{attribute 'GeneratedUsingTerminal: EL6002-0000-0016'}
{attribute addProperty BoxType "EL6002-0000-0016"}
{attribute addProperty Id "EtcSlaveTerminalBaseCOM_Inputs_Channel_1AT %I*COM_Inputs_Channel_3801C95E30COM_Inputs_Channel_2AT %I*COM_Inputs_Channel_3801C95E30COM_Outputs_Channel_1AT %Q*COM_Outputs_Channel_EADA2E0D27COM_Outputs_Channel_2AT %Q*COM_Outputs_Channel_EADA2E0D27WcStateAT %I*WcState_9091E0EB2InfoDataAT %I*InfoData_32EB74EA10"}
{attribute addProperty CRC "2353564961"}
{attribute addProperty Size "126"}
TYPE EL6002_8C488D21 EXTENDS EtcSlaveTerminalBase :
STRUCT
	{attribute addProperty Name "COM_Inputs_Channel_1"}
	COM_Inputs_Channel_1 : COM_Inputs_Channel_3801C95E;
	{attribute addProperty Name "COM_Inputs_Channel_2"}
	COM_Inputs_Channel_2 : COM_Inputs_Channel_3801C95E;
	{attribute addProperty Name "COM_Outputs_Channel_1"}
	COM_Outputs_Channel_1 : COM_Outputs_Channel_EADA2E0D;
	{attribute addProperty Name "COM_Outputs_Channel_2"}
	COM_Outputs_Channel_2 : COM_Outputs_Channel_EADA2E0D;
	{attribute addProperty Name "WcState"}
	WcState : WcState_9091E0EB;
	{attribute addProperty Name "InfoData"}
	InfoData : InfoData_32EB74EA;
END_STRUCT
END_TYPE

(* stored: Version 1.2.0.0, ProductVersion 3.1.4024.9
   DUT EL6002_8C488D21: Id {e8473469-5dd8-4e42-9c70-8c86456dc9c8} *)
